(*
    Estados possíveis do ciclo automático do Exercício 06.
    PARADO  -> máquina ociosa, aguardando comando de ligar.
    AVANCA  -> ferramenta avançando até a posição de trabalho.
    AGUARDA -> tempo de espera na posição de trabalho (simula operação).
    RECUA   -> ferramenta recuando à posição de repouso.
*)
TYPE E_EstadoCiclo :
(
	PARADO,
	AVANCA,
	AGUARDA,
	RECUA
);
END_TYPE

(* stored: Version 1.1.0.1
   DUT E_EstadoCiclo: Id {a1b2c3d4-0001-4002-8002-000000000006} *)
